// TIA Portal V20 export
VAR_GLOBAL   // PLC tag table "00_Simulation"
END_VAR
